Universal Robots PolyScope program: p2_Group1_v3.urp

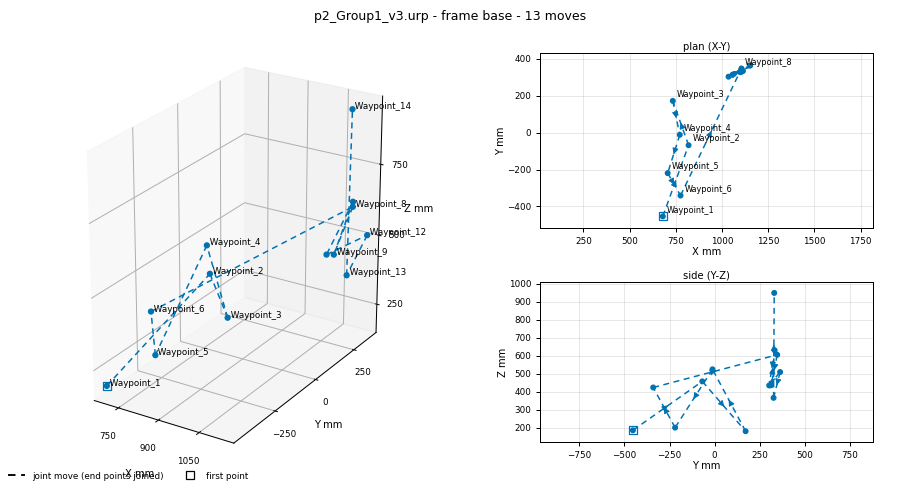
[picture p0: tool path of p2_Group1_v3.urp in frame base, 13 of 13 moves have a stored position in this frame; points joined in program order, loops and branches not executed]
Program p2_Group1_v3 (installation=default directory=/programs/usbdisk/Project2_v3 createdIn=5.13.0 lastSavedIn=5.13.0 robotSerialNumber=20225201357)
Calibrated DH parameters: a=[-0.000097, -0.065329, -0.560646, 0.000001, -0.00004, 0]; d=[0.180831, -263.113709, 285.24385, -21.955837, 0.119737, 0.115719]; alpha=[1.571643, -0.002312, 0.004975, 1.569542, -1.570894, 0]; deltaTheta=[0, 1.463798, 5.013296, -0.193909, 0, 0]
InitVariablesNode
Robot Program (runOnlyOnce=false)
  robotState := read_port_register(200)
  If robotState≟0
    MoveJ speed 60 deg/s, acceleration 80 deg/s^2 (useActiveTCP=true) feature=Base
      Waypoint Waypoint_1: TCP in base x=679.966 y=-453.337 z=186.367 mm, rx=-0.167 ry=0.3103 rz=0.6326 rad; joints [-21.071, -102.748, -100.738, -63.17, 89.355, 31.664] deg; TCP offset x=-0.19 y=3.58 z=256.26 mm, rx=0.0015 ry=-2.7841 rz=0 rad
      Waypoint Waypoint_2: TCP in base x=819.328 y=-68.464 z=457.654 mm, rx=-0.3031 ry=-0.0982 rz=1.074 rad; joints [4.934, -88.987, -95.041, -63.1, 95.517, 30.877] deg
      Waypoint Waypoint_3: TCP in base x=733.911 y=171.658 z=181.321 mm, rx=-0.0736 ry=-0.0404 rz=1.3818 rad; joints [19.025, -95.43, -114.898, -45.931, 105.167, 30.894] deg
      Waypoint Waypoint_4: TCP in base x=771.734 y=-11.897 z=524.446 mm, rx=-0.5897 ry=0.052 rz=1.2099 rad; joints [18.943, -83.124, -93.069, -74.524, 76.464, 30.893] deg
      Waypoint Waypoint_5: TCP in base x=706.283 y=-219.357 z=201.134 mm, rx=-0.5627 ry=0.5407 rz=1.0955 rad; joints [8.026, -94.837, -110.077, -68.051, 67.72, 30.913] deg
      Waypoint Waypoint_6: TCP in base x=775.842 y=-340.758 z=423.774 mm, rx=-0.479 ry=0.2817 rz=0.8271 rad; joints [-5.811, -94.458, -89.362, -74.274, 76.64, 30.91] deg
  ElseIf robotState≟1
    MoveJ speed 60 deg/s, acceleration 80 deg/s^2 (useActiveTCP=true) feature=Base
      Waypoint Waypoint_8: TCP in base x=1105.662 y=346.84 z=605.108 mm, rx=-1.0601 ry=-0.7242 rz=1.2732 rad; joints [33.261, -108.549, -82.99, -13.989, 67.349, 11.84] deg
      Waypoint Waypoint_9: TCP in base x=1057.2 y=312.981 z=436.038 mm, rx=-0.9757 ry=-0.2822 rz=1.5339 rad; joints [33.217, -108.526, -84.67, -38.239, 67.362, 11.844] deg
      Waypoint Waypoint_10: TCP in base x=1113.447 y=332.965 z=629.595 mm, rx=-1.0708 ry=-0.6582 rz=1.2856 rad; joints [32.826, -108.553, -78.783, -21.122, 66.141, 11.693] deg
      Waypoint Waypoint_11: TCP in base x=1035.618 y=302.486 z=435.006 mm, rx=-0.9108 ry=-0.1421 rz=1.6189 rad; joints [32.82, -108.557, -79.928, -51.542, 69.111, 11.807] deg
      Waypoint Waypoint_12: TCP in base x=1152.714 y=362.931 z=509.455 mm, rx=-1.0455 ry=-0.6011 rz=1.3385 rad; joints [32.7, -115.157, -79.1, -18.204, 67.187, 11.805] deg
      Waypoint Waypoint_13: TCP in base x=1099.289 y=326.761 z=366.268 mm, rx=-0.9625 ry=-0.2094 rz=1.5583 rad; joints [32.66, -115.172, -80.503, -39.553, 67.195, 11.807] deg
      Waypoint Waypoint_14: TCP in base x=1105.422 y=330.367 z=948.035 mm, rx=-1.1195 ry=-1.4315 rz=0.665 rad; joints [32.663, -115.164, -66.779, 22.948, 66.716, 11.808] deg
